Yaskawa INFORM job: frame_planes_program.JBI

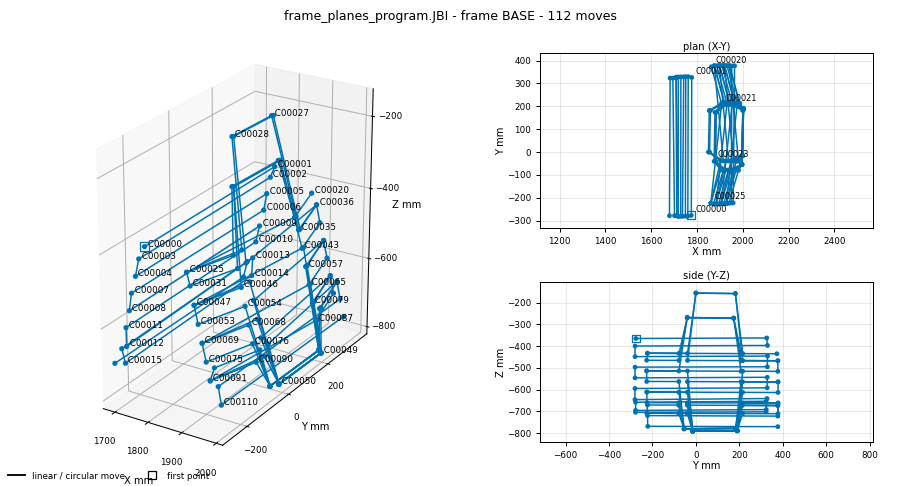
[picture p0: tool path of frame_planes_program.JBI in frame BASE, 112 of 115 moves have a stored position in this frame; points joined in program order, loops and branches not executed]
/JOB
//NAME frame_planes_program
//POS
///NPOS 112,0,112,0,0,0
///TOOL 0
///POSTYPE BASE
///RECTAN
///RCONF 0,0,0,0,0,0,0,0,0,0,0,0,0,0,0,0,0,0,0,0,0,0,0,0
C00000=1775.255312,-276.613391,-364.487959,175.000000,-77.692921,-5.000000
C00001=1777.150757,325.985194,-362.060651,175.000000,-77.692921,-5.000000
C00002=1761.744575,329.398619,-396.655085,175.000000,-77.692921,-5.000000
C00003=1760.026199,-280.205061,-399.154050,175.000000,-77.692921,-5.000000
C00004=1749.328660,-280.338953,-447.997463,175.000000,-77.692921,-5.000000
C00005=1751.156731,329.443068,-445.521589,175.000000,-77.692921,-5.000000
C00006=1742.172443,328.813964,-494.741108,175.000000,-77.692921,-5.000000
C00007=1736.645304,-280.458414,-496.407574,175.000000,-77.692921,-5.000000
C00008=1728.931130,-280.404901,-545.900968,175.000000,-77.692921,-5.000000
C00009=1729.727517,328.554100,-543.203897,175.000000,-77.692921,-5.000000
C00010=1718.336783,328.065063,-591.897754,175.000000,-77.692921,-5.000000
C00011=1717.928117,-280.650264,-594.678263,175.000000,-77.692921,-5.000000
C00012=1718.698335,-280.769134,-646.023464,175.000000,-77.692921,-5.000000
C00013=1709.052043,327.554030,-641.051168,175.000000,-77.692921,-5.000000
C00014=1708.238529,323.881760,-692.067606,175.000000,-77.692921,-5.000000
C00015=1711.748752,-277.770716,-695.669782,175.000000,-77.692921,-5.000000
C00016=1701.859800,-277.835606,-658.086735,175.000000,-77.692921,-5.000000
C00017=1694.576612,323.454209,-653.663141,175.000000,-77.692921,-5.000000
C00018=1682.749762,323.216773,-702.260667,175.000000,-77.692921,-5.000000
C00019=1679.812094,-278.068120,-704.454408,180.000000,-60.000000,0.000000
C00020=1862.881325,372.686708,-434.795355,-5.000000,-77.568322,175.000000
C00021=1908.206670,208.414035,-434.137283,5.000000,-89.838880,133.626946
C00022=1878.669814,173.956558,-271.700446,175.000000,-63.416141,-33.303256
C00023=1875.034198,-39.997217,-269.150022,-175.000000,-62.451422,29.753952
C00024=1902.833779,-77.955216,-432.975013,-175.000000,-89.832276,43.626474
C00025=1860.563483,-223.242344,-432.378276,175.000000,-90.000000,5.000000
C00026=1908.234399,215.543653,-434.166201,5.000000,-89.838880,133.626946
C00027=1853.683385,181.644232,-158.256094,175.000000,-63.416137,-33.303370
C00028=1850.172542,-0.084100,-155.836676,-175.000000,-62.451523,29.753905
C00029=1902.986848,-38.599676,-433.134638,-175.000000,-89.832276,43.626474
C00030=1860.563483,-223.242344,-432.378276,175.000000,-90.000000,5.000000
C00031=1872.486897,-226.667838,-464.802182,-5.000000,-77.568322,175.000000
C00032=1915.042518,-78.048107,-465.368746,-175.000000,-89.844395,43.588761
C00033=1879.892619,-39.969316,-268.118680,175.000000,-62.472861,29.733721
C00034=1883.719927,173.985608,-270.550625,175.000000,-63.396078,-33.324707
C00035=1920.653026,208.317989,-466.447746,-5.000000,-89.850324,133.589168
C00036=1875.631773,377.299896,-467.076435,175.000000,-90.000000,5.000000
C00037=1915.247444,-38.692568,-465.516940,175.000000,-89.844395,43.588761
C00038=1855.082919,-0.056297,-154.793686,175.000000,-62.472860,29.733754
C00039=1858.741975,181.673055,-157.104606,-175.000000,-63.396189,-33.324666
C00040=1920.690151,215.447607,-466.474593,-5.000000,-89.850324,133.589168
C00041=1875.631773,377.299896,-467.076435,175.000000,-90.000000,5.000000
C00042=1886.575653,377.260542,-515.864795,-5.000000,-77.568322,175.000000
C00043=1931.683965,208.057043,-515.220307,5.000000,-89.846795,133.600813
C00044=1883.994442,173.976715,-270.501417,-175.000000,-63.402278,-33.318119
C00045=1880.225948,-39.977883,-268.033122,175.000000,-62.466330,29.739916
C00046=1926.146705,-78.310038,-514.115637,175.000000,-89.840661,43.600387
C00047=1883.675541,-226.823008,-513.536017,175.000000,-90.000000,5.000000
C00048=1931.718193,215.186661,-515.247792,-5.000000,-89.846795,133.600813
C00049=2001.892638,189.932626,-789.606820,5.000000,-58.406621,138.441476
C00050=1997.714778,-14.960801,-791.421455,5.000000,-57.515812,-141.907852
C00051=1926.335645,-38.954498,-514.267355,175.000000,-89.840661,43.600387
C00052=1883.675541,-226.823008,-513.536017,175.000000,-90.000000,5.000000
C00053=1894.757040,-226.550131,-562.295575,-5.000000,-77.568322,175.000000
C00054=1937.469947,-78.485757,-562.834367,175.000000,-89.851536,43.566512
C00055=1995.719269,-54.222704,-780.317567,5.000000,-57.524693,-141.935636
C00056=2000.237862,182.896254,-778.644151,5.000000,-58.399046,138.413063
C00057=1943.220632,207.878428,-563.864246,-5.000000,-89.857082,133.566883
C00058=1898.374910,378.005593,-564.468448,175.000000,-90.000000,5.000000
C00059=1937.705464,-39.130217,-562.975817,-175.000000,-89.851536,43.566512
C00060=1998.335592,-14.920647,-791.254807,5.000000,-57.524596,-141.935331
C00061=2002.659720,189.972773,-789.465259,5.000000,-58.399147,138.413331
C00062=1943.263298,215.008046,-563.889871,-5.000000,-89.857082,133.566883
C00063=1898.374910,378.005593,-564.468448,175.000000,-90.000000,5.000000
C00064=1909.541036,378.140180,-613.208670,-5.000000,-77.568322,175.000000
C00065=1954.261790,207.667629,-612.624106,-5.000000,-89.861975,133.550761
C00066=2000.508480,182.915381,-778.597676,-5.000000,-58.395463,138.399636
C00067=1995.901777,-54.203442,-780.263095,5.000000,-57.528888,-141.948802
C00068=1948.409693,-78.695148,-611.629764,-175.000000,-89.856700,43.550416
C00069=1905.586588,-225.895389,-611.112550,175.000000,-90.000000,5.000000
C00070=1954.308466,214.797248,-612.648847,5.000000,-89.861975,133.550761
C00071=2002.934839,189.992398,-789.418108,5.000000,-58.395481,138.399561
C00072=1998.538866,-14.900775,-791.195302,5.000000,-57.528925,-141.948915
C00073=1948.667342,-39.339608,-611.766335,175.000000,-89.856700,43.550416
C00074=1905.586588,-225.895389,-611.112550,175.000000,-90.000000,5.000000
C00075=1916.792329,-225.466543,-659.845485,-5.000000,-77.568322,175.000000
C00076=1959.526510,-78.957454,-660.373798,175.000000,-89.852910,43.562232
C00077=1996.250632,-54.217763,-780.196849,5.000000,-57.525742,-141.939000
C00078=2000.791669,182.901044,-778.525460,-5.000000,-58.398114,138.409682
C00079=1965.304164,207.406358,-661.394226,5.000000,-89.858383,133.562595
C00080=1920.494977,378.170158,-661.995154,175.000000,-90.000000,5.000000
C00081=1959.767913,-39.601915,-660.513950,175.000000,-89.852910,43.562232
C00082=1998.870887,-14.914902,-791.132617,-5.000000,-57.525825,-141.939247
C00083=2003.215202,189.978174,-789.346544,-5.000000,-58.398129,138.409538
C00084=1965.347897,214.535976,-661.419616,5.000000,-89.858383,133.562595
C00085=1920.494977,378.170158,-661.995154,175.000000,-90.000000,5.000000
C00086=1931.360347,378.143042,-710.800882,-5.000000,-77.568322,175.000000
C00087=1976.287962,207.138111,-710.178708,5.000000,-89.853623,133.578289
C00088=2001.019298,182.882764,-778.462875,5.000000,-58.401466,138.422472
C00089=1996.561911,-54.235800,-780.141716,5.000000,-57.521756,-141.926640
C00090=1970.609023,-79.227057,-709.123687,-175.000000,-89.847882,43.577900
C00091=1927.989091,-225.322918,-708.578999,175.000000,-90.000000,5.000000
C00092=1976.327791,214.267729,-710.204958,5.000000,-89.853623,133.578289
C00093=2003.438118,189.959299,-789.284480,5.000000,-58.401634,138.422767
C00094=1999.162788,-14.933910,-791.082459,5.000000,-57.521633,-141.926226
C00095=1970.828883,-39.871517,-709.268589,-175.000000,-89.847882,43.577900
C00096=1927.989091,-225.322918,-708.578999,175.000000,-90.000000,5.000000
C00097=1939.246219,-223.257114,-670.706109,-5.000000,-77.568322,175.000000
C00098=1981.539665,-79.551104,-671.291777,175.000000,-89.833612,43.622319
C00099=1996.710582,-54.288028,-780.148291,5.000000,-57.510103,-141.890775
C00100=2000.926938,182.830205,-778.447897,-5.000000,-58.410982,138.459160
C00101=1986.938734,206.817805,-672.444873,5.000000,-89.840140,133.622783
C00102=1941.668826,377.207894,-673.122371,175.000000,-90.000000,5.000000
C00103=1981.698447,-40.195564,-671.450143,-175.000000,-89.833612,43.622319
C00104=1999.249074,-14.985513,-791.102137,-5.000000,-57.510188,-141.890824
C00105=2003.335860,189.907729,-789.271830,-5.000000,-58.411168,138.458872
C00106=1986.967499,213.947423,-672.473563,5.000000,-89.840140,133.622783
C00107=1941.668826,377.207894,-673.122371,175.000000,-90.000000,5.000000
C00108=1952.358286,377.016313,-721.966069,-5.000000,-77.568322,175.000000
C00109=1949.674528,-222.751005,-719.610804,-5.000000,-77.568322,175.000000
C00110=1958.005294,-221.860436,-768.979778,-5.000000,-77.568322,175.000000
C00111=1964.425148,377.250442,-770.508219,180.000000,-60.000000,0.000000
///POSTYPE PULSE
///PULSE
EC00000=90112.0
EC00001=90112.0
EC00002=90112.0
EC00003=90112.0
EC00004=90112.0
EC00005=90112.0
EC00006=90112.0
EC00007=90112.0
EC00008=90112.0
EC00009=90112.0
EC00010=90112.0
EC00011=90112.0
EC00012=90112.0
EC00013=90112.0
EC00014=90112.0
EC00015=90112.0
EC00016=90112.0
EC00017=90112.0
EC00018=90112.0
EC00019=90112.0
EC00020=273408.0
EC00021=273408.0
EC00022=273408.0
EC00023=273408.0
EC00024=273408.0
EC00025=273408.0
EC00026=273408.0
EC00027=273408.0
EC00028=273408.0
EC00029=273408.0
EC00030=273408.0
EC00031=273408.0
EC00032=273408.0
EC00033=273408.0
EC00034=273408.0
EC00035=273408.0
EC00036=273408.0
EC00037=273408.0
EC00038=273408.0
EC00039=273408.0
EC00040=273408.0
EC00041=273408.0
EC00042=273408.0
EC00043=273408.0
EC00044=273408.0
EC00045=273408.0
EC00046=273408.0
EC00047=273408.0
EC00048=273408.0
EC00049=273408.0
EC00050=273408.0
EC00051=273408.0
EC00052=273408.0
EC00053=273408.0
EC00054=273408.0
EC00055=273408.0
EC00056=273408.0
EC00057=273408.0
EC00058=273408.0
EC00059=273408.0
EC00060=273408.0
EC00061=273408.0
EC00062=273408.0
EC00063=273408.0
EC00064=273408.0
EC00065=273408.0
EC00066=273408.0
EC00067=273408.0
EC00068=273408.0
EC00069=273408.0
EC00070=273408.0
EC00071=273408.0
EC00072=273408.0
EC00073=273408.0
EC00074=273408.0
EC00075=273408.0
EC00076=273408.0
EC00077=273408.0
EC00078=273408.0
EC00079=273408.0
EC00080=273408.0
EC00081=273408.0
EC00082=273408.0
EC00083=273408.0
EC00084=273408.0
EC00085=273408.0
EC00086=273408.0
EC00087=273408.0
EC00088=273408.0
EC00089=273408.0
EC00090=273408.0
EC00091=273408.0
EC00092=273408.0
EC00093=273408.0
EC00094=273408.0
EC00095=273408.0
EC00096=273408.0
EC00097=273408.0
EC00098=273408.0
EC00099=273408.0
EC00100=273408.0
EC00101=273408.0
EC00102=273408.0
EC00103=273408.0
EC00104=273408.0
EC00105=273408.0
EC00106=273408.0
EC00107=273408.0
EC00108=273408.0
EC00109=273408.0
EC00110=273408.0
EC00111=273408.0
//INST
///DATE 2023/08/16 15:18
///ATTR SC,RW,RJ
////FRAME BASE
///GROUP1 RB1,ST1
NOP
MOVJ P009 EX000 VJ=15.00
MOVJ C00000 EC00000 VJ=15.0
CALL JOB:SPYON
MOVL C00001 EC00001 V=150.0
MOVL C00002 EC00002 V=150.0
MOVL C00003 EC00003 V=150.0
MOVL C00004 EC00004 V=150.0
MOVL C00005 EC00005 V=150.0
MOVL C00006 EC00006 V=150.0
MOVL C00007 EC00007 V=150.0
MOVL C00008 EC00008 V=150.0
MOVL C00009 EC00009 V=150.0
MOVL C00010 EC00010 V=150.0
MOVL C00011 EC00011 V=150.0
MOVL C00012 EC00012 V=150.0
MOVL C00013 EC00013 V=150.0
MOVL C00014 EC00014 V=150.0
MOVL C00015 EC00015 V=150.0
MOVL C00016 EC00016 V=150.0
MOVL C00017 EC00017 V=150.0
MOVL C00018 EC00018 V=150.0
MOVL C00019 EC00019 V=150.0
CALL JOB:SPYOF
MOVJ P009 VJ=15.00
MOVJ C00020 EC00020 VJ=15.0
CALL JOB:SPYON
MOVL C00021 EC00021 V=150.0
MOVL C00022 EC00022 V=150.0
MOVL C00023 EC00023 V=150.0
MOVL C00024 EC00024 V=150.0
MOVL C00025 EC00025 V=150.0
MOVL C00026 EC00026 V=150.0
MOVL C00027 EC00027 V=150.0
MOVL C00028 EC00028 V=150.0
MOVL C00029 EC00029 V=150.0
MOVL C00030 EC00030 V=150.0
MOVL C00031 EC00031 V=150.0
MOVL C00032 EC00032 V=150.0
MOVL C00033 EC00033 V=150.0
MOVL C00034 EC00034 V=150.0
MOVL C00035 EC00035 V=150.0
MOVL C00036 EC00036 V=150.0
MOVL C00037 EC00037 V=150.0
MOVL C00038 EC00038 V=150.0
MOVL C00039 EC00039 V=150.0
MOVL C00040 EC00040 V=150.0
MOVL C00041 EC00041 V=150.0
MOVL C00042 EC00042 V=150.0
MOVL C00043 EC00043 V=150.0
MOVL C00044 EC00044 V=150.0
MOVL C00045 EC00045 V=150.0
MOVL C00046 EC00046 V=150.0
MOVL C00047 EC00047 V=150.0
MOVL C00048 EC00048 V=150.0
MOVL C00049 EC00049 V=150.0
MOVL C00050 EC00050 V=150.0
MOVL C00051 EC00051 V=150.0
MOVL C00052 EC00052 V=150.0
MOVL C00053 EC00053 V=150.0
MOVL C00054 EC00054 V=150.0
MOVL C00055 EC00055 V=150.0
MOVL C00056 EC00056 V=150.0
MOVL C00057 EC00057 V=150.0
MOVL C00058 EC00058 V=150.0
MOVL C00059 EC00059 V=150.0
MOVL C00060 EC00060 V=150.0
MOVL C00061 EC00061 V=150.0
MOVL C00062 EC00062 V=150.0
MOVL C00063 EC00063 V=150.0
MOVL C00064 EC00064 V=150.0
MOVL C00065 EC00065 V=150.0
MOVL C00066 EC00066 V=150.0
MOVL C00067 EC00067 V=150.0
MOVL C00068 EC00068 V=150.0
MOVL C00069 EC00069 V=150.0
MOVL C00070 EC00070 V=150.0
MOVL C00071 EC00071 V=150.0
MOVL C00072 EC00072 V=150.0
MOVL C00073 EC00073 V=150.0
MOVL C00074 EC00074 V=150.0
MOVL C00075 EC00075 V=150.0
MOVL C00076 EC00076 V=150.0
MOVL C00077 EC00077 V=150.0
MOVL C00078 EC00078 V=150.0
MOVL C00079 EC00079 V=150.0
MOVL C00080 EC00080 V=150.0
MOVL C00081 EC00081 V=150.0
MOVL C00082 EC00082 V=150.0
MOVL C00083 EC00083 V=150.0
MOVL C00084 EC00084 V=150.0
MOVL C00085 EC00085 V=150.0
MOVL C00086 EC00086 V=150.0
MOVL C00087 EC00087 V=150.0
MOVL C00088 EC00088 V=150.0
MOVL C00089 EC00089 V=150.0
MOVL C00090 EC00090 V=150.0
MOVL C00091 EC00091 V=150.0
MOVL C00092 EC00092 V=150.0
MOVL C00093 EC00093 V=150.0
MOVL C00094 EC00094 V=150.0
MOVL C00095 EC00095 V=150.0
MOVL C00096 EC00096 V=150.0
MOVL C00097 EC00097 V=150.0
MOVL C00098 EC00098 V=150.0
MOVL C00099 EC00099 V=150.0
MOVL C00100 EC00100 V=150.0
MOVL C00101 EC00101 V=150.0
MOVL C00102 EC00102 V=150.0
MOVL C00103 EC00103 V=150.0
MOVL C00104 EC00104 V=150.0
MOVL C00105 EC00105 V=150.0
MOVL C00106 EC00106 V=150.0
MOVL C00107 EC00107 V=150.0
MOVL C00108 EC00108 V=150.0
MOVL C00109 EC00109 V=150.0
MOVL C00110 EC00110 V=150.0
MOVL C00111 EC00111 V=150.0
CALL JOB:SPYOF
MOVJ P009 VJ=15.00
END
